// TIA Portal V21 export
// export: Created 2026-07-07T09:15:55.8352405Z, ExportSetting WithReadOnly, DisplayName Totally Integrated Automation Portal, DisplayVersion V21, DisplayName SINAMICS Startdrive Advanced, DisplayVersion V21, DisplayName SINAMICS Startdrive G110M, G120, G120C, G120D, G120P, G115D, DisplayVersion V21, DisplayName SINAMICS Startdrive G130, G150, S120, S150, G200, G220, S200, S210, S220, Innomotics MVD, DisplayVersion V21, DisplayName STEP 7 Professional, DisplayVersion V21, DisplayName STEP 7 Safety, DisplayVersion V21, DisplayName Tech WebApplication, DisplayVersion V21, DisplayName WinCC Basic/Comfort/Advanced, DisplayVersion V21, DisplayName WinCC Professional, DisplayVersion V21, DisplayName WinCC Unified, DisplayVersion V21
Screen "根画面"  Nonex480, Template=模板_1
  on GenerateScreen: SetTag(Tag := Tag_ScreenNumber, Value := 1)
  ScreenLayer 
    TextField "HmiScreenItemData" at 80,226 size 640x22  Text="欢迎进入 HMI_1 (KTP900 Basic+ PN)！"
